INTERFACE PUBLIC OutputStream EXTENDS __System.IQueryInterface

METHOD PUBLIC Close
END_METHOD

METHOD PUBLIC Flush
END_METHOD

METHOD Write : BOOL
VAR_INPUT
	data : BYTE;
END_VAR
END_METHOD

END_INTERFACE

(* stored: Version 1.1.0.1
   Itf OutputStream: Id {956022d5-1c24-4fb3-bfec-21bc3da876e8}
   Method Close: Id {29b22d46-831e-4c2e-879b-c0ebbee3d884}
   Method Flush: Id {8ecbba24-7588-4fb2-be59-726d55ae5a11}
   Method Write: Id {310641f9-105a-40a3-aedc-65afd4ed324c} *)
